PROGRAM A26
VAR_IN_OUT
	spacerRecollector : SpacerRecollectionUnit;
END_VAR
VAR
	robot7 : RobotA26; //placeholder, will need another robot definition for A26
	robotSliderA26 : ServoNC;
END_VAR
VAR //sensors to detect spacer on transfer conveyors
	spacerPresent_A24_LRC_C02 AT %I* : BOOL;
	spacerPresent_A24_LRC_C04 AT %I* : BOOL;
	spacerPresent_A24_LRC_C06 AT %I* : BOOL;
	spacerPresent_A24_LRC_C08 AT %I* : BOOL;
	spacerPresent_A24_LRC_C10 AT %I* : BOOL;
	spacerPresent_A24_LRC_C12 AT %I* : BOOL;
END_VAR

callHardware();
setupHardware();
runModules();
callHardware();

METHOD PRIVATE callHardware : BOOL
VAR_INPUT
END_VAR
robot7();	
robotSliderA26(bEnable:= TRUE, ready=> , position=> , velocity=> );
END_METHOD

METHOD PRIVATE runModules : BOOL
VAR_INPUT
END_VAR
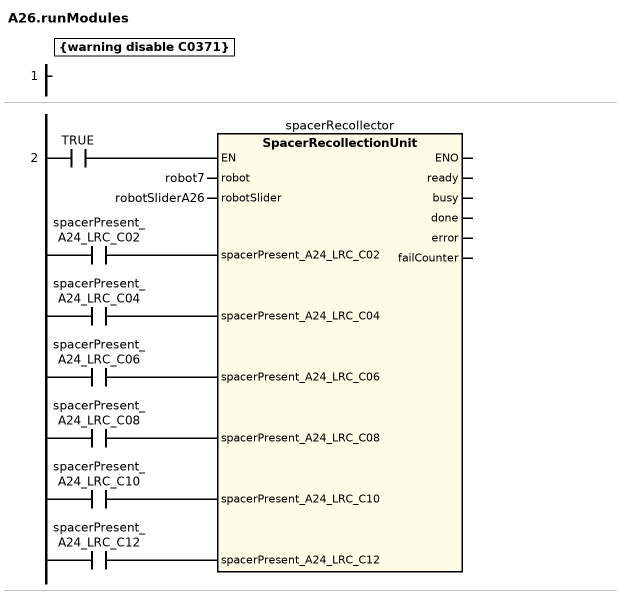
// NETWORK 1
// label: {warning disable C0371}

// NETWORK 2
spacerRecollector(
    robot := robot7,
    robotSlider := robotSliderA26,
    spacerPresent_A24_LRC_C02 := spacerPresent_A24_LRC_C02,
    spacerPresent_A24_LRC_C04 := spacerPresent_A24_LRC_C04,
    spacerPresent_A24_LRC_C06 := spacerPresent_A24_LRC_C06,
    spacerPresent_A24_LRC_C08 := spacerPresent_A24_LRC_C08,
    spacerPresent_A24_LRC_C10 := spacerPresent_A24_LRC_C10,
    spacerPresent_A24_LRC_C12 := spacerPresent_A24_LRC_C12); // SpacerRecollectionUnit
END_METHOD

METHOD PRIVATE setupHardware : BOOL
VAR
	iCornerGuardSlot : CornerGuard;
	iCardboardSlot : Cardboard;
	i : INT;
END_VAR
END_METHOD

END_PROGRAM

(* stored: Version 1.1.0.1, ProductVersion 3.1.4024.11
   POU A26: Id {df70bd72-3010-4603-acfe-2b41c91cc9fb}, SpecialFunc None
   Method callHardware: Id {28545458-26ff-4a6a-af8e-aff99ab2b072}
   Method runModules: Id {91fb3897-d479-41a4-ac07-1d36f5ff9718}
   Method setupHardware: Id {0b0eb0a5-de16-4ffc-920a-53d441a1c49c} *)
